Staubli VAL3: GetAppVersion.pgx

program GetAppVersion(string& answer)
begin
//*******************************************************************************
//*   ______
//*  / _____) /|
//* | |      / /
//* | | /\  / /
//* | | \ \/ /  _      Copyright (c) KEOLABS, 2016
//* | |  \__/  | |        http://www.keolabs.com
//* | |________| |
//*  \__________/
//*
//********************************************************************************
//*@file          : GetAppVersion
//*@author        : Yves Ragot
//*@version       : $Id: GetAppVersion.pgx 1645 2017-01-24 08:09:09Z yves $
//*@brief         : Get firmware version (application version)
//*******************************************************************************/

  answer = "v1.1 jan 23 2017"

end
